{attribute 'GeneratedUsingTerminal: EPP3204-0002-0016'}
{attribute addProperty BoxType "EPP3204-0002-0016"}
{attribute addProperty Description "EPP3204-0002 4Ch. Ana. Input PT100 (RTD)"}
{attribute addProperty Physics "YY"}
{attribute addProperty Id "RTD_RTDInputs_Channel_1AT %I*RTD_RTDInputs_Channel_A8DF64E310RTD_RTDInputs_Channel_2AT %I*RTD_RTDInputs_Channel_A8DF64E310RTD_RTDInputs_Channel_3AT %I*RTD_RTDInputs_Channel_A8DF64E310RTD_RTDInputs_Channel_4AT %I*RTD_RTDInputs_Channel_A8DF64E310WcStateAT %I*WcState_9091E0EB2InfoDataAT %I*InfoData_32EB74EA10"}
{attribute addProperty CRC "1826087193"}
{attribute addProperty Size "52"}
TYPE EPP3204_6CD7E119 EXTENDS EtcSlaveBoxBase_77A0E4A7 :
STRUCT
	{attribute addProperty Name "RTD_RTDInputs_Channel_1"}
	RTD_RTDInputs_Channel_1 : RTD_RTDInputs_Channel_A8DF64E3;
	{attribute addProperty Name "RTD_RTDInputs_Channel_2"}
	RTD_RTDInputs_Channel_2 : RTD_RTDInputs_Channel_A8DF64E3;
	{attribute addProperty Name "RTD_RTDInputs_Channel_3"}
	RTD_RTDInputs_Channel_3 : RTD_RTDInputs_Channel_A8DF64E3;
	{attribute addProperty Name "RTD_RTDInputs_Channel_4"}
	RTD_RTDInputs_Channel_4 : RTD_RTDInputs_Channel_A8DF64E3;
	{attribute addProperty Name "WcState"}
	WcState : WcState_9091E0EB;
	{attribute addProperty Name "InfoData"}
	InfoData : InfoData_32EB74EA;
END_STRUCT
END_TYPE

(* stored: Version 1.2.0.0, ProductVersion 3.1.4024.11
   DUT EPP3204_6CD7E119: Id {4dae3cdf-a5ad-45ad-82d8-a5857d1c76b6} *)
